KUKA KRL data list: LoadSensing.dat

&ACCESS RVO4
DEFDAT CenterOfMass_EVAL PUBLIC
;FOLD EXTERNAL DECLARATIONS;%{PE}%MKUKATPBASIS,%CEXT,%VCOMMON,%P
;FOLD BASISTECH EXT;%{PE}%MKUKATPBASIS,%CEXT,%VEXT,%P
EXT  BAS (BAS_COMMAND  :IN,REAL  :IN )
;ENDFOLD (BASISTECH EXT)
;FOLD USER EXT;%{E}%MKUKATPUSER,%CEXT,%VEXT,%P
;Make your modifications here

; Center of gravity coordinates (F/T sensor reference frame)
DECL GLOBAL REAL POS_CG[3]
DECL GLOBAL REAL TOOL_WEIGHT

;F0 & T0
DECL GLOBAL REAL myF0[3]
DECL GLOBAL REAL myM0[3]

;F/T sensor data (sampled from the PLC and streamed to the KRC4 via EtheCAT bus)
SIGNAL Fx $IN[513] TO $IN[544]
SIGNAL Fy $IN[545] TO $IN[576]
SIGNAL Fz $IN[577] TO $IN[608]
SIGNAL Tx $IN[609] TO $IN[640]
SIGNAL Ty $IN[641] TO $IN[672]
SIGNAL Tz $IN[673] TO $IN[704]

;ENDFOLD (USER EXT)
;ENDFOLD (EXTERNAL DECLARATIONS)
ENDDAT
